FUNCTION_BLOCK FB_Integrate
// This FB increments the value of the Input with every call of the FB. DO NOT CALL THIS TWICE IN A CYCLE.
// Integration is done with the trapeze method
// The Reset input resets the value to 0
VAR_INPUT
	IN_DataToIntegrate		: REAL;
	IN_CmdReset				: BOOL;
	
END_VAR
VAR_OUTPUT
	OUT_IntegrationValue	: REAL;
END_VAR
VAR
	OldData					: REAL;
	OldTime					: TIME;
	DeltaTime				: TIME;
END_VAR

IF OldTime > T#0S THEN
	DeltaTime := TIME()-OldTime;
	
	OUT_IntegrationValue := OUT_IntegrationValue+(IN_DataToIntegrate + OldData)*TIME_TO_REAL(DeltaTime)/2000.0;
	
	OldTime := TIME();
	OldData := IN_DataToIntegrate;
	
	IF IN_CmdReset THEN
		OUT_IntegrationValue := 0.0;
		OldData := 0.0;
	END_IF
ELSE
	OldTime := TIME();
	OldData := IN_DataToIntegrate;
END_IF

END_FUNCTION_BLOCK

(* stored: Version 1.1.0.1, ProductVersion 3.1.4024.6
   POU FB_Integrate: Id {69486986-b944-4910-bc43-be5f9427bd94}, SpecialFunc None *)
